{attribute 'qualified_only'}
VAR_GLOBAL
	
	newUser			: STRING;
	newUserGroup	: STRING;
	newUserAutoL	: STRING;
	newUserPassword	: STRING;
	
END_VAR

(* stored: Version 1.1.0.1, ProductVersion 3.1.4024.12
   GVL GVL_UserManagement: Id {499b15c8-e412-485d-8222-f042dddda31d} *)
